// TIA Portal V20 export
TYPE "OutPut"
   STRUCT
      Active : Bool;   // Roller is Active
      TrfInSetRdyRcv : Bool;   // Ready to Receive: Signal to previous object set
      TrfInSetArrived : Bool;   // Body Arrived: Signal to previous object Set
      TrfInSetActive : Bool;   // Transfer in set active
      TrfInSetFinished : Bool;   // Transfer in set finished
      TrfOutSetRdyDlv : Bool;   // Ready to Deliver: Signal to next object set
      TrfOutSetTM : Bool;   // Transfer: Signal to next object set
      TrfOutSetActive : Bool;   // Transfer out set active
      TrfOutSetFinished : Bool;   // Transfer out set finished
      TrfInResRdyRcv : Bool;   // Ready to Receive: Signal to previous object Reset
      TrfInResArrived : Bool;   // Body Arrived: Signal to previous object Reset
      TrfInResActive : Bool;   // Transfer in Reset active
      TrfInResFinished : Bool;   // Transfer in Reset finished
      TrfOutResRdyDlv : Bool;   // Ready to Deliver: Signal to next object Reset
      TrfOutResTM : Bool;   // Transfer: Signal to next object Reset
      TrfOutResActive : Bool;   // Transfer out Reset active
      TrfOutResFinished : Bool;   // Transfer out Reset finished
      BodyInPosition : Bool;   // Body In Position / Body in Position on roller
      NoSkid : Bool;   // No Skid
      LSpdSet : Bool;   // Lower Speed Set
      HSpdSet : Bool;   // Hight Speed Set
      SelectLower : Bool;   // Selext Lower Speed
   END_STRUCT;
END_TYPE
